// TIA Portal V20 export
// export: Created 2026-04-11T06:02:30.7528608Z, ExportSetting WithDefaults, DisplayName Totally Integrated Automation Portal, DisplayVersion V20, DisplayName TIA Portal Openness, DisplayVersion V20, DisplayName TIA Portal Version Control Interface, DisplayVersion V20, DisplayName STEP 7 Professional, DisplayVersion V20, DisplayName STEP 7 Safety, DisplayVersion V20, DisplayName WinCC Basic/Comfort/Advanced, DisplayVersion V20, DisplayName WinCC Unified, DisplayVersion V20
TYPE "udtHandshakes"
// stored: IsFailsafeCompliant false
   STRUCT
      bDelivering { ExternalWritable := 'False'} : Bool;   // Delivery in progress
      bSystemReady { ExternalWritable := 'False'} : Bool;   // System not ready for selection
      iSelected { ExternalWritable := 'False'} : Int;   // Currently selected queue item
      rActual { ExternalWritable := 'False'} : Real;   // Delivered actual value
      Handshake { ExternalWritable := 'False'; S7_SetPoint := 'True'} : Array[1.."Handshakes.iSize"] of "udtHandshake";   // Requests array
   END_STRUCT;
END_TYPE
